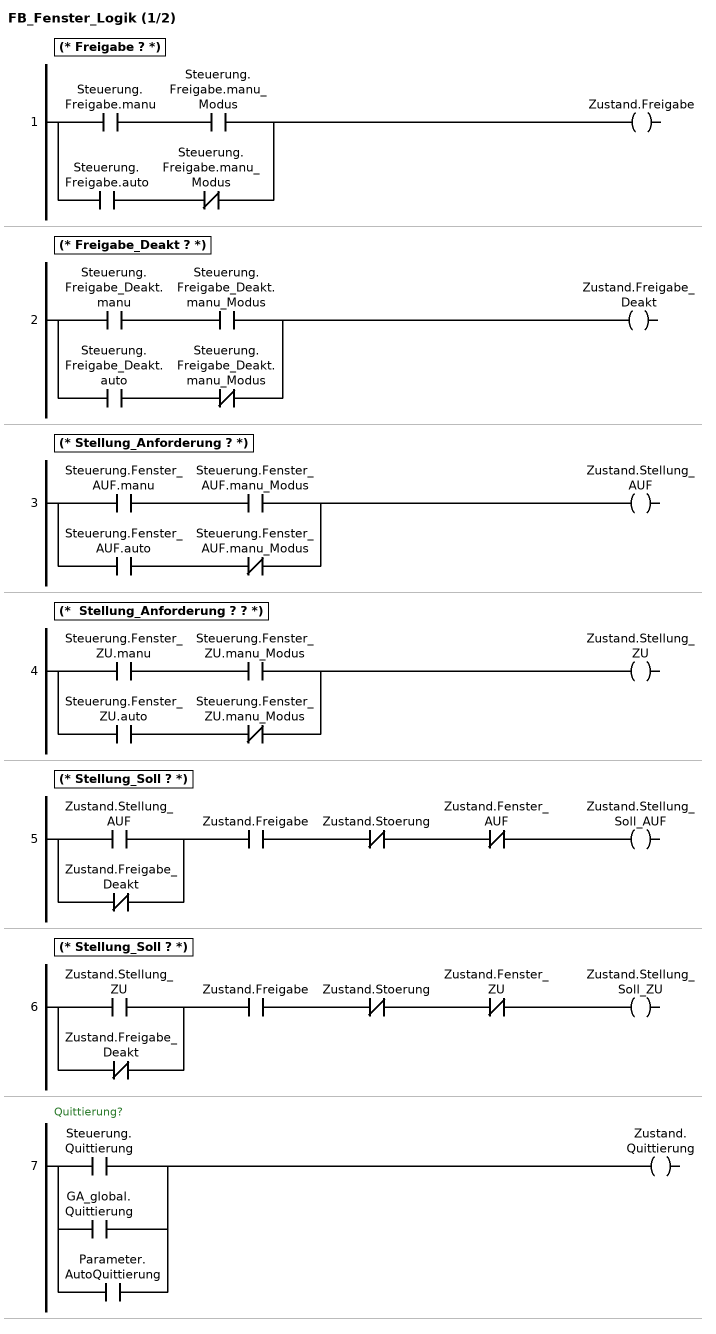
// NETWORK 1
// label: (* Freigabe ? *)
Zustand.Freigabe := Steuerung.Freigabe.manu AND Steuerung.Freigabe.manu_Modus OR Steuerung.Freigabe.auto AND NOT Steuerung.Freigabe.manu_Modus;

// NETWORK 2
// label: (* Freigabe_Deakt ? *)
Zustand.Freigabe_Deakt := Steuerung.Freigabe_Deakt.manu AND Steuerung.Freigabe_Deakt.manu_Modus OR Steuerung.Freigabe_Deakt.auto AND NOT Steuerung.Freigabe_Deakt.manu_Modus;

// NETWORK 3
// label: (* Stellung_Anforderung ? *)
Zustand.Stellung_AUF := Steuerung.Fenster_AUF.manu AND Steuerung.Fenster_AUF.manu_Modus OR Steuerung.Fenster_AUF.auto AND NOT Steuerung.Fenster_AUF.manu_Modus;

// NETWORK 4
// label: (*  Stellung_Anforderung ? ? *)
Zustand.Stellung_ZU := Steuerung.Fenster_ZU.manu AND Steuerung.Fenster_ZU.manu_Modus OR Steuerung.Fenster_ZU.auto AND NOT Steuerung.Fenster_ZU.manu_Modus;

// NETWORK 5
// label: (* Stellung_Soll ? *)
Zustand.Stellung_Soll_AUF := (Zustand.Stellung_AUF OR NOT Zustand.Freigabe_Deakt) AND Zustand.Freigabe AND NOT Zustand.Stoerung AND NOT Zustand.Fenster_AUF;

// NETWORK 6
// label: (* Stellung_Soll ? *)
Zustand.Stellung_Soll_ZU := (Zustand.Stellung_ZU OR NOT Zustand.Freigabe_Deakt) AND Zustand.Freigabe AND NOT Zustand.Stoerung AND NOT Zustand.Fenster_ZU;

// NETWORK 7
// Quittierung?
Zustand.Quittierung := Steuerung.Quittierung OR GA_global.Quittierung OR Parameter.AutoQuittierung;

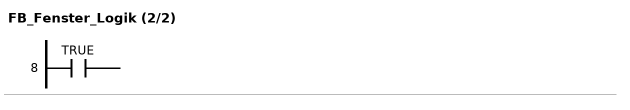
// NETWORK 8

END_FUNCTION_BLOCK

// ---- POUs/Einzelanlagen/RGBW-Kanal/FB_RGBW_Zustandscheck.TcPOU
FUNCTION_BLOCK FB_RGBW_Zustandscheck
VAR_INPUT
	Zustand		: ST_RGBW_Zustand;
	Steuerung	: ST_RGBW_Steuerung;
END_VAR
VAR_OUTPUT
END_VAR
VAR
	RGB_Werte	: ARRAY[0..2] OF BYTE;
	TGB_Werte	: BOOL;
END_VAR

IF Zustand.Betrieb THEN
	HEXSTR_TO_DATA(Steuerung.Farbcode, ADR(RGB_Werte), SIZEOF(RGB_Werte));
	Zustand.R_Wert 	:= RGB_Werte[0];
	Zustand.G_Wert	:= RGB_Werte[1];
	Zustand.B_Wert	:= RGB_Werte[2];
	(*Zustand.W_Wert	:= (0.2126 * ((Zustand.R_Wert / 255) ** 2.2) + 0.7152 * ((Zustand.G_Wert / 255) ** 2.2) + 0.0722 * ((Zustand.B_Wert / 255) ** 2.2));*)
ELSE
	Zustand.R_Wert 	:= 0;
	Zustand.G_Wert	:= 0;
	Zustand.B_Wert	:= 0;
	Zustand.W_Wert	:= 0;
END_IF;

END_FUNCTION_BLOCK

// ---- POUs/Einzelanlagen/Stromzähler/ABB_Stromzaehler/FB_ABB_Lesen.TcPOU
FUNCTION_BLOCK FB_ABB_Lesen
VAR_INPUT
	Reg1Value	: LREAL;
	Reg42Value	: LREAL;
	Reg42Unit 	: STRING;
END_VAR
VAR_OUTPUT
	Arbeit 		: LREAL;
	Leistung 	: LREAL;
	CosPhi		: LREAL;
	(*Scheinleistung: LREAL;
	Blindleistung: LREAL;*)
END_VAR
VAR
	Telegram 	: INT;
END_VAR

(*Der Zähler sendet 5 Versch. Diagramme, es werden jedoch von der Klemme immer nur 2 Diagramme gelesen. Durch prüfen der Einheit des Registers 42 kann bestimmt werden welches Diagramm aktuell gelesen wird.
Reg42.sUnit = 'W' --> Telegram 1+2 werden aktuell ausgelesen
Reg42.sUnit = 'Wh' --> Telegram 3+4 werden aktuell ausgelesen
Reg42.sUnit = '' --> Telegram 5 wird aktuell ausgelesen
*)

IF REG42Unit = 'W' THEN
	Telegram :=1;
ELSIF REG42Unit = 'Wh' THEN
	Telegram :=3;
ELSIF REG42Unit = '' THEN
	Telegram :=5;
END_IF

CASE Telegram OF
	1: 	Arbeit := Reg1Value;
		Leistung := Reg42Value;
	3:	CosPhi := Reg1Value/INT_TO_LREAL(1000);
END_CASE;

(*
(*Scheinleistung berechnen, abfangen von div by 0 error*)
IF  CosPhi<>0  THEN
Scheinleistung := Leistung/CosPhi;
END_IF

(*Blindleistung aus geom Summe berechen, abfangen einer "negativen Wurzel")*)
IF Scheinleistung>Blindleistung THEN
Blindleistung := SQRT(Scheinleistung*Scheinleistung-Leistung*Leistung);
END_IF
*)

END_FUNCTION_BLOCK

// ---- POUs/Einzelanlagen/Stromzähler/ABB_Stromzaehler/FB_Stromzaehler_BHKW.TcPOU
FUNCTION_BLOCK FB_Stromzaehler_BHKW
VAR_INPUT
	Telegramm	: ARRAY[1..cMBUS_MaxTelegrams] OF ST_MBus_Data2;

END_VAR
VAR_IN_OUT
	Zustand		: ST_SZ_Zustand;
END_VAR
VAR
END_VAR
VAR // added by the converter: edge detectors and wires of the graphical bodies
    _w1, _w2 : ANY;
END_VAR

Zustand.Arbeit := _w1;
Zustand.Leistung := _w2;
_w1 := STRING_TO_REAL(Telegramm[1].arrData[1].sValue);
_w2 := STRING_TO_REAL(Telegramm[1].arrData[2].sValue);

END_FUNCTION_BLOCK

// ---- POUs/Einzelanlagen/Stromzähler/ABB_Stromzaehler/FB_Stromzaehler_Gebaeude.TcPOU
FUNCTION_BLOCK FB_Stromzaehler_Gebaeude
VAR_INPUT
	Telegramm	: ARRAY[1..cMBUS_MaxTelegrams] OF ST_MBus_Data2;
END_VAR
VAR_IN_OUT
	Zustand		: ST_SZ_Zustand;
END_VAR
VAR
	Leistungsberechnung			: FB_ABB_Lesen;
END_VAR
VAR // added by the converter: edge detectors and wires of the graphical bodies
    _w1 : ANY;
END_VAR

Zustand.Arbeit := STRING_TO_REAL(Telegramm[1].arrData[1].sValue);
Zustand.Leistung := STRING_TO_REAL(Telegramm[2].arrData[2].sValue);
Zustand.Leistungsfaktor := _w1;
_w1 := STRING_TO_REAL(Telegramm[1].arrData[3].sValue) / 1000;

END_FUNCTION_BLOCK

// ---- POUs/Einzelanlagen/Stromzähler/Netzanschlusspunkt/FB_Stromzaehler_NSHV_Modbus.TcPOU
FUNCTION_BLOCK FB_Stromzaehler_NSHV_Modbus
VAR_IN_OUT
	Stromzaehler_NSHV	: ST_NSHV_Zustand;
END_VAR
VAR_OUTPUT
END_VAR
VAR
	MB_KM				:	ARRAY[1..1] OF ST_NSHV_Modbus;
	ModbusAddress	 	: ARRAY [1..1] OF BYTE := [1]; (*Modbusadressen der beiden Geräte*)
	FtrigBusy			: F_TRIG;
	Timeout 			: TIME := T#300ms;		(* timeout while waiting for an answer of the modbus slave *)
	Unit				: BYTE;
	state				: INT;
	busy				: BOOL;
	LetzterFehlerState	: INT;
	LetzterModbusFehler	: ST_ModbusErrorDiagnostics;
	CounterError		: DINT;
	CounterSuccess		: DINT;
	NSHV_Wert_zuweisen	: FB_NSHV_Wert_zuweisen;
END_VAR

CASE state OF
	0:
		Modbus_NSHV.ReadRegs(Execute:= FALSE); (* Initialisierung*)
		Modbus_NSHV.WriteRegs(Execute:= FALSE);

		(*Auswahl von Modbus-Slaves 1 und 2*)
		Unit := Unit + 1;
		IF Unit  >1 THEN
			Unit := 1;
		END_IF

		state := state + 1;


	1:	(*= NSHV_Spannung_PH1_N lesen =*)
		Modbus_NSHV.ReadRegs(
				UnitID:= ModbusAddress[Unit], (* station address *)
				Quantity:= 2, (*Datenwörter *)
				MBAddr:= 16#1002,
				cbLength:= SIZEOF(MB_KM[Unit].Modbus_Adresse1[16#1002]),
				pMemoryAddr:= ADR(MB_KM[Unit].Modbus_Adresse1[16#1002]),
				Execute:= TRUE,
				Timeout:= Timeout,
				Busy => busy	);
			IF NOT busy THEN
				Modbus_NSHV.ReadRegs(Execute:= FALSE);
				IF Modbus_NSHV.Error THEN
					MB_KM[Unit].Modbus_Unit_Online := FALSE; (*Modbus Gerät ist offline*)
					state := 0;
				ELSE
					MB_KM[Unit].Modbus_Unit_Online := TRUE; (*Modbus Gerät ist online*)
					state := state + 1;
				END_IF
			END_IF


	2:	(*= NSHV_Spannung_PH2_N lesen =*)
		Modbus_NSHV.ReadRegs(
				UnitID:= ModbusAddress[Unit], (* station address *)
				Quantity:= 2, (*Datenwörter *)
				MBAddr:= 16#1004,
				cbLength:= SIZEOF(MB_KM[Unit].Modbus_Adresse1[16#1004]),
				pMemoryAddr:= ADR(MB_KM[Unit].Modbus_Adresse1[16#1004]),
				Execute:= TRUE,
				Timeout:= Timeout,
				Busy => busy	);
			IF NOT busy THEN
				Modbus_NSHV.ReadRegs(Execute:= FALSE);
				IF Modbus_NSHV.Error THEN
					MB_KM[Unit].Modbus_Unit_Online := FALSE; (*Modbus Gerät ist offline*)
					state := 0;
				ELSE
					MB_KM[Unit].Modbus_Unit_Online := TRUE; (*Modbus Gerät ist online*)
					state := state + 1;
				END_IF
			END_IF


	3:	(*= NSHV_Spannung_PH3_N lesen =*)
		Modbus_NSHV.ReadRegs(
				UnitID:= ModbusAddress[Unit], (* station address *)
				Quantity:= 2, (*Datenwörter *)
				MBAddr:= 16#1006,
				cbLength:= SIZEOF(MB_KM[Unit].Modbus_Adresse1[16#1006]),
				pMemoryAddr:= ADR(MB_KM[Unit].Modbus_Adresse1[16#1006]),
				Execute:= TRUE,
				Timeout:= Timeout,
				Busy => busy	);
			IF NOT busy THEN
				Modbus_NSHV.ReadRegs(Execute:= FALSE);
				IF Modbus_NSHV.Error THEN
					MB_KM[Unit].Modbus_Unit_Online := FALSE; (*Modbus Gerät ist offline*)
					state := 0;
				ELSE
					MB_KM[Unit].Modbus_Unit_Online := TRUE; (*Modbus Gerät ist online*)
					state := state + 1;
				END_IF
			END_IF


	4:	(*= NSHV_Strom_PH1 lesen =*)
		Modbus_NSHV.ReadRegs(
				UnitID:= ModbusAddress[Unit], (* station address *)
				Quantity:= 2, (*Datenwörter *)
				MBAddr:= 16#1010,
				cbLength:= SIZEOF(MB_KM[Unit].Modbus_Adresse1[16#1010]),
				pMemoryAddr:= ADR(MB_KM[Unit].Modbus_Adresse1[16#1010]),
				Execute:= TRUE,
				Timeout:= Timeout,
				Busy => busy	);
			IF NOT busy THEN
				Modbus_NSHV.ReadRegs(Execute:= FALSE);
				IF Modbus_NSHV.Error THEN
					MB_KM[Unit].Modbus_Unit_Online := FALSE; (*Modbus Gerät ist offline*)
					state := 0;
				ELSE
					MB_KM[Unit].Modbus_Unit_Online := TRUE; (*Modbus Gerät ist online*)
					state := state + 1;
				END_IF
			END_IF


	5:	(*= NSHV_Strom_PH2 lesen =*)
		Modbus_NSHV.ReadRegs(
				UnitID:= ModbusAddress[Unit], (* station address *)
				Quantity:= 2, (*Datenwörter *)
				MBAddr:= 16#1012,
				cbLength:= SIZEOF(MB_KM[Unit].Modbus_Adresse1[16#1012]),
				pMemoryAddr:= ADR(MB_KM[Unit].Modbus_Adresse1[16#1012]),
				Execute:= TRUE,
				Timeout:= Timeout,
				Busy => busy	);
			IF NOT busy THEN
				Modbus_NSHV.ReadRegs(Execute:= FALSE);
				IF Modbus_NSHV.Error THEN
					MB_KM[Unit].Modbus_Unit_Online := FALSE; (*Modbus Gerät ist offline*)
					state := 0;
				ELSE
					MB_KM[Unit].Modbus_Unit_Online := TRUE; (*Modbus Gerät ist online*)
					state := state + 1;
				END_IF
			END_IF

	6:	(*= NSHV_Strom_PH3 lesen =*)
		Modbus_NSHV.ReadRegs(
				UnitID:= ModbusAddress[Unit], (* station address *)
				Quantity:= 2, (*Datenwörter *)
				MBAddr:= 16#1014,
				cbLength:= SIZEOF(MB_KM[Unit].Modbus_Adresse1[16#1014]),
				pMemoryAddr:= ADR(MB_KM[Unit].Modbus_Adresse1[16#1014]),
				Execute:= TRUE,
				Timeout:= Timeout,
				Busy => busy	);
			IF NOT busy THEN
				Modbus_NSHV.ReadRegs(Execute:= FALSE);
				IF Modbus_NSHV.Error THEN
					MB_KM[Unit].Modbus_Unit_Online := FALSE; (*Modbus Gerät ist offline*)
					state := 0;
				ELSE
					MB_KM[Unit].Modbus_Unit_Online := TRUE; (*Modbus Gerät ist online*)
					state := state + 1;
				END_IF
			END_IF


	7:	(*= NSHV_Wirkleistung lesen =*)
		Modbus_NSHV.ReadRegs(
				UnitID:= ModbusAddress[Unit], (* station address *)
				Quantity:= 2, (*Datenwörter *)
				MBAddr:= 16#102E,
				cbLength:= SIZEOF(MB_KM[Unit].Modbus_Adresse1[16#102E]),
				pMemoryAddr:= ADR(MB_KM[Unit].Modbus_Adresse1[16#102E]),
				Execute:= TRUE,
				Timeout:= Timeout,
				Busy => busy	);
			IF NOT busy THEN
				Modbus_NSHV.ReadRegs(Execute:= FALSE);
				IF Modbus_NSHV.Error THEN
					MB_KM[Unit].Modbus_Unit_Online := FALSE; (*Modbus Gerät ist offline*)
					state := 0;
				ELSE
					MB_KM[Unit].Modbus_Unit_Online := TRUE; (*Modbus Gerät ist online*)
					state := state + 1;
				END_IF
			END_IF

	8:	(*= NSHV_Blindleistung lesen =*)
		Modbus_NSHV.ReadRegs(
				UnitID:= ModbusAddress[Unit], (* station address *)
				Quantity:= 2, (*Datenwörter *)
				MBAddr:= 16#1036,
				cbLength:= SIZEOF(MB_KM[Unit].Modbus_Adresse1[16#1036]),
				pMemoryAddr:= ADR(MB_KM[Unit].Modbus_Adresse1[16#1036]),
				Execute:= TRUE,
				Timeout:= Timeout,
				Busy => busy	);
			IF NOT busy THEN
				Modbus_NSHV.ReadRegs(Execute:= FALSE);
				IF Modbus_NSHV.Error THEN
					MB_KM[Unit].Modbus_Unit_Online := FALSE; (*Modbus Gerät ist offline*)
					state := 0;
				ELSE
					MB_KM[Unit].Modbus_Unit_Online := TRUE; (*Modbus Gerät ist online*)
					state := state + 1;
				END_IF
			END_IF


	9:	(*= NSHV_Scheinleistung lesen =*)
		Modbus_NSHV.ReadRegs(
				UnitID:= ModbusAddress[Unit], (* station address *)
				Quantity:= 2, (*Datenwörter *)
				MBAddr:= 16#1026,
				cbLength:= SIZEOF(MB_KM[Unit].Modbus_Adresse1[16#1026]),
				pMemoryAddr:= ADR(MB_KM[Unit].Modbus_Adresse1[16#1026]),
				Execute:= TRUE,
				Timeout:= Timeout,
				Busy => busy	);
			IF NOT busy THEN
				Modbus_NSHV.ReadRegs(Execute:= FALSE);
				IF Modbus_NSHV.Error THEN
					MB_KM[Unit].Modbus_Unit_Online := FALSE; (*Modbus Gerät ist offline*)
					state := 0;
				ELSE
					MB_KM[Unit].Modbus_Unit_Online := TRUE; (*Modbus Gerät ist online*)
					state := state + 1;
				END_IF
			END_IF

	10:	(*= NSHV_Frequenz lesen =*)
		Modbus_NSHV.ReadRegs(
				UnitID:= ModbusAddress[Unit], (* station address *)
				Quantity:= 2, (*Datenwörter *)
				MBAddr:= 16#1046,
				cbLength:= SIZEOF(MB_KM[Unit].Modbus_Adresse1[16#1046]),
				pMemoryAddr:= ADR(MB_KM[Unit].Modbus_Adresse1[16#1046]),
				Execute:= TRUE,
				Timeout:= Timeout,
				Busy => busy	);
			IF NOT busy THEN
				Modbus_NSHV.ReadRegs(Execute:= FALSE);
				IF Modbus_NSHV.Error THEN
					MB_KM[Unit].Modbus_Unit_Online := FALSE; (*Modbus Gerät ist offline*)
					state := 0;
				ELSE
					MB_KM[Unit].Modbus_Unit_Online := TRUE; (*Modbus Gerät ist online*)
					state := state + 1;
				END_IF
			END_IF

	11:	(*= NSHV_Harmonische_Verzerrung_U_PH1_THD lesen =*)
		Modbus_NSHV.ReadRegs(
				UnitID:= ModbusAddress[Unit], (* station address *)
				Quantity:= 2, (*Datenwörter *)
				MBAddr:= 16#1048,
				cbLength:= SIZEOF(MB_KM[Unit].Modbus_Adresse1[16#1048]),
				pMemoryAddr:= ADR(MB_KM[Unit].Modbus_Adresse1[16#1048]),
				Execute:= TRUE,
				Timeout:= Timeout,
				Busy => busy	);
			IF NOT busy THEN
				Modbus_NSHV.ReadRegs(Execute:= FALSE);
				IF Modbus_NSHV.Error THEN
					MB_KM[Unit].Modbus_Unit_Online := FALSE; (*Modbus Gerät ist offline*)
					state := 0;
				ELSE
					MB_KM[Unit].Modbus_Unit_Online := TRUE; (*Modbus Gerät ist online*)
					state := state + 1;
				END_IF
			END_IF

	12:	(*= NSHV_Harmonische_Verzerrung_U_PH2_THD lesen =*)
		Modbus_NSHV.ReadRegs(
				UnitID:= ModbusAddress[Unit], (* station address *)
				Quantity:= 2, (*Datenwörter *)
				MBAddr:= 16#104A,
				cbLength:= SIZEOF(MB_KM[Unit].Modbus_Adresse1[16#104A]),
				pMemoryAddr:= ADR(MB_KM[Unit].Modbus_Adresse1[16#104A]),
				Execute:= TRUE,
				Timeout:= Timeout,
				Busy => busy	);
			IF NOT busy THEN
				Modbus_NSHV.ReadRegs(Execute:= FALSE);
				IF Modbus_NSHV.Error THEN
					MB_KM[Unit].Modbus_Unit_Online := FALSE; (*Modbus Gerät ist offline*)
					state := 0;
				ELSE
					MB_KM[Unit].Modbus_Unit_Online := TRUE; (*Modbus Gerät ist online*)
					state := state + 1;
				END_IF
			END_IF

	13:	(*= NSHV_Harmonische_Verzerrung_U_PH3_THD lesen =*)
		Modbus_NSHV.ReadRegs(
				UnitID:= ModbusAddress[Unit], (* station address *)
				Quantity:= 2, (*Datenwörter *)
				MBAddr:= 16#104C,
				cbLength:= SIZEOF(MB_KM[Unit].Modbus_Adresse1[16#104C]),
				pMemoryAddr:= ADR(MB_KM[Unit].Modbus_Adresse1[16#104C]),
				Execute:= TRUE,
				Timeout:= Timeout,
				Busy => busy	);
			IF NOT busy THEN
				Modbus_NSHV.ReadRegs(Execute:= FALSE);
				IF Modbus_NSHV.Error THEN
					MB_KM[Unit].Modbus_Unit_Online := FALSE; (*Modbus Gerät ist offline*)
					state := 0;
				ELSE
					MB_KM[Unit].Modbus_Unit_Online := TRUE; (*Modbus Gerät ist online*)
					state := state + 1;
				END_IF
			END_IF

	14:	(*= NSHV_Harmonische_Verzerrung_I_PH1_THD lesen =*)
		Modbus_NSHV.ReadRegs(
				UnitID:= ModbusAddress[Unit], (* station address *)
				Quantity:= 2, (*Datenwörter *)
				MBAddr:= 16#104E,
				cbLength:= SIZEOF(MB_KM[Unit].Modbus_Adresse1[16#104E]),
				pMemoryAddr:= ADR(MB_KM[Unit].Modbus_Adresse1[16#104E]),
				Execute:= TRUE,
				Timeout:= Timeout,
				Busy => busy	);
			IF NOT busy THEN
				Modbus_NSHV.ReadRegs(Execute:= FALSE);
				IF Modbus_NSHV.Error THEN
					MB_KM[Unit].Modbus_Unit_Online := FALSE; (*Modbus Gerät ist offline*)
					state := 0;
				ELSE
					MB_KM[Unit].Modbus_Unit_Online := TRUE; (*Modbus Gerät ist online*)
					state := state + 1;
				END_IF
			END_IF

	15:	(*= NSHV_Harmonische_Verzerrung_I_PH2_THD lesen =*)
		Modbus_NSHV.ReadRegs(
				UnitID:= ModbusAddress[Unit], (* station address *)
				Quantity:= 2, (*Datenwörter *)
				MBAddr:= 16#1050,
				cbLength:= SIZEOF(MB_KM[Unit].Modbus_Adresse1[16#1050]),
				pMemoryAddr:= ADR(MB_KM[Unit].Modbus_Adresse1[16#1050]),
				Execute:= TRUE,
				Timeout:= Timeout,
				Busy => busy	);
			IF NOT busy THEN
				Modbus_NSHV.ReadRegs(Execute:= FALSE);
				IF Modbus_NSHV.Error THEN
					MB_KM[Unit].Modbus_Unit_Online := FALSE; (*Modbus Gerät ist offline*)
					state := 0;
				ELSE
					MB_KM[Unit].Modbus_Unit_Online := TRUE; (*Modbus Gerät ist online*)
					state := state + 1;
				END_IF
			END_IF

	16:	(*= NSHV_Harmonische_Verzerrung_I_PH3_THD lesen =*)
		Modbus_NSHV.ReadRegs(
				UnitID:= ModbusAddress[Unit], (* station address *)
				Quantity:= 2, (*Datenwörter *)
				MBAddr:= 16#1052,
				cbLength:= SIZEOF(MB_KM[Unit].Modbus_Adresse1[16#1052]),
				pMemoryAddr:= ADR(MB_KM[Unit].Modbus_Adresse1[16#1052]),
				Execute:= TRUE,
				Timeout:= Timeout,
				Busy => busy	);
			IF NOT busy THEN
				Modbus_NSHV.ReadRegs(Execute:= FALSE);
				IF Modbus_NSHV.Error THEN
					MB_KM[Unit].Modbus_Unit_Online := FALSE; (*Modbus Gerät ist offline*)
					state := 0;
				ELSE
					MB_KM[Unit].Modbus_Unit_Online := TRUE; (*Modbus Gerät ist online*)
					state := state + 1;
				END_IF
			END_IF

	17:	(*= NSHV_Importierte_Wirkenergie lesen =*)
			Modbus_NSHV.ReadRegs(
					UnitID:= ModbusAddress[Unit], (* station address *)
					Quantity:= 2, (*Datenwörter *)
					MBAddr:= 16#103E,
					cbLength:= SIZEOF(MB_KM[Unit].Modbus_Adresse1[16#103E]),
					pMemoryAddr:= ADR(MB_KM[Unit].Modbus_Adresse1[16#103E]),
					Execute:= TRUE,
					Timeout:= Timeout,
					Busy => busy	);
				IF NOT busy THEN
					Modbus_NSHV.ReadRegs(Execute:= FALSE);
					IF Modbus_NSHV.Error THEN
						MB_KM[Unit].Modbus_Unit_Online := FALSE; (*Modbus Gerät ist offline*)
						state := 0;
					ELSE
						MB_KM[Unit].Modbus_Unit_Online := TRUE; (*Modbus Gerät ist online*)
						state := state + 1;
					END_IF
				END_IF

	18:	(*= NSHV_Exportierte_Wirkenergie lesen =*)
			Modbus_NSHV.ReadRegs(
					UnitID:= ModbusAddress[Unit], (* station address *)
					Quantity:= 2, (*Datenwörter *)
					MBAddr:= 16#1042,
					cbLength:= SIZEOF(MB_KM[Unit].Modbus_Adresse1[16#1042]),
					pMemoryAddr:= ADR(MB_KM[Unit].Modbus_Adresse1[16#1042]),
					Execute:= TRUE,
					Timeout:= Timeout,
					Busy => busy	);
				IF NOT busy THEN
					Modbus_NSHV.ReadRegs(Execute:= FALSE);
					IF Modbus_NSHV.Error THEN
						MB_KM[Unit].Modbus_Unit_Online := FALSE; (*Modbus Gerät ist offline*)
						state := 0;
					ELSE
						MB_KM[Unit].Modbus_Unit_Online := TRUE; (*Modbus Gerät ist online*)
						state := state + 1;
					END_IF
				END_IF

	19:	(*= NSHV_Max_LN_Wirkleistung_Demand lesen =*)
			Modbus_NSHV.ReadRegs(
					UnitID:= ModbusAddress[Unit], (* station address *)
					Quantity:= 2, (*Datenwörter *)
					MBAddr:= 16#1070,
					cbLength:= SIZEOF(MB_KM[Unit].Modbus_Adresse1[16#1070]),
					pMemoryAddr:= ADR(MB_KM[Unit].Modbus_Adresse1[16#1070]),
					Execute:= TRUE,
					Timeout:= Timeout,
					Busy => busy	);
				IF NOT busy THEN
					Modbus_NSHV.ReadRegs(Execute:= FALSE);
					IF Modbus_NSHV.Error THEN
						MB_KM[Unit].Modbus_Unit_Online := FALSE; (*Modbus Gerät ist offline*)
						state := 0;
					ELSE
						MB_KM[Unit].Modbus_Unit_Online := TRUE; (*Modbus Gerät ist online*)
						state := 0;
					END_IF
				END_IF
END_CASE

(*Zählen von erfolgreichen und fehlgeschlagenen Leseversuchen*)
FtrigBusy(CLK:=Modbus_NSHV.BUSY );
IF FtrigBusy.Q THEN
	IF Modbus_NSHV.Error THEN
		LetzterModbusFehler := Modbus_NSHV.ErrorDiagnostics;
		LetzterFehlerState := state;
		CounterError := CounterError + 1;
	ELSE
		CounterSuccess := CounterSuccess + 1;
	END_IF
END_IF

(* Zuweisen der Modbus-Werte zu den Zaehler Variablen *)

NSHV_Wert_zuweisen(Input:= MB_KM[1].Modbus_Adresse1[16#1002], Output => Stromzaehler_NSHV.Spannung_Ph1_N);
NSHV_Wert_zuweisen(Input:= MB_KM[1].Modbus_Adresse1[16#1004], Output => Stromzaehler_NSHV.Spannung_Ph2_N);
NSHV_Wert_zuweisen(Input:= MB_KM[1].Modbus_Adresse1[16#1006], Output => Stromzaehler_NSHV.Spannung_Ph3_N);

NSHV_Wert_zuweisen(Input:= MB_KM[1].Modbus_Adresse1[16#1010], Output => Stromzaehler_NSHV.Strom_Ph1);
NSHV_Wert_zuweisen(Input:= MB_KM[1].Modbus_Adresse1[16#1012], Output => Stromzaehler_NSHV.Strom_Ph2);
NSHV_Wert_zuweisen(Input:= MB_KM[1].Modbus_Adresse1[16#1014], Output => Stromzaehler_NSHV.Strom_Ph3);

NSHV_Wert_zuweisen(Input:= MB_KM[1].Modbus_Adresse1[16#102E], Output => Stromzaehler_NSHV.Wirkleistung);
NSHV_Wert_zuweisen(Input:= MB_KM[1].Modbus_Adresse1[16#1036], Output => Stromzaehler_NSHV.Blindleistung);
NSHV_Wert_zuweisen(Input:= MB_KM[1].Modbus_Adresse1[16#1026], Output => Stromzaehler_NSHV.Scheinleistung);
NSHV_Wert_zuweisen(Input:= MB_KM[1].Modbus_Adresse1[16#1046], Output => Stromzaehler_NSHV.Frequenz);

NSHV_Wert_zuweisen(Input:= MB_KM[1].Modbus_Adresse1[16#1048], Output => Stromzaehler_NSHV.Harmonische_Verzerrung_U_Ph1_THD);
NSHV_Wert_zuweisen(Input:= MB_KM[1].Modbus_Adresse1[16#104A], Output => Stromzaehler_NSHV.Harmonische_Verzerrung_U_Ph2_THD);
NSHV_Wert_zuweisen(Input:= MB_KM[1].Modbus_Adresse1[16#104C], Output => Stromzaehler_NSHV.Harmonische_Verzerrung_U_Ph3_THD );
NSHV_Wert_zuweisen(Input:= MB_KM[1].Modbus_Adresse1[16#104E], Output => Stromzaehler_NSHV.Harmonische_Verzerrung_I_Ph1_THD);
NSHV_Wert_zuweisen(Input:= MB_KM[1].Modbus_Adresse1[16#1050], Output => Stromzaehler_NSHV.Harmonische_Verzerrung_I_Ph2_THD);
NSHV_Wert_zuweisen(Input:= MB_KM[1].Modbus_Adresse1[16#1052], Output => Stromzaehler_NSHV.Harmonische_Verzerrung_I_Ph3_THD);

NSHV_Wert_zuweisen(Input:= MB_KM[1].Modbus_Adresse1[16#103E], Output => Stromzaehler_NSHV.Importierte_Wirkenergie);
NSHV_Wert_zuweisen(Input:= MB_KM[1].Modbus_Adresse1[16#1042], Output => Stromzaehler_NSHV.Exportierte_Wirkenergie);
NSHV_Wert_zuweisen(Input:= MB_KM[1].Modbus_Adresse1[16#1070], Output => Stromzaehler_NSHV.Max_Wirkleistung_Demand_System );



Stromzaehler_NSHV.Stoerung := NOT MB_KM[1].Modbus_Unit_Online;

END_FUNCTION_BLOCK

// ---- POUs/Einzelanlagen/Waermepumpe/FB_WP_Ablaufsteuerung.TcPOU
FUNCTION_BLOCK FB_WP_Ablaufsteuerung
VAR_IN_OUT
	Zustand			: ST_WP_Zustand;
	Stellwert		: ST_WP_Stellwert;
END_VAR
VAR_INPUT
	Steuerung		: ST_WP_Steuerung;
	Parameter		: ST_WP_Parameter;
END_VAR
VAR_OUTPUT
END_VAR
VAR
	Timer			: TON;
END_VAR

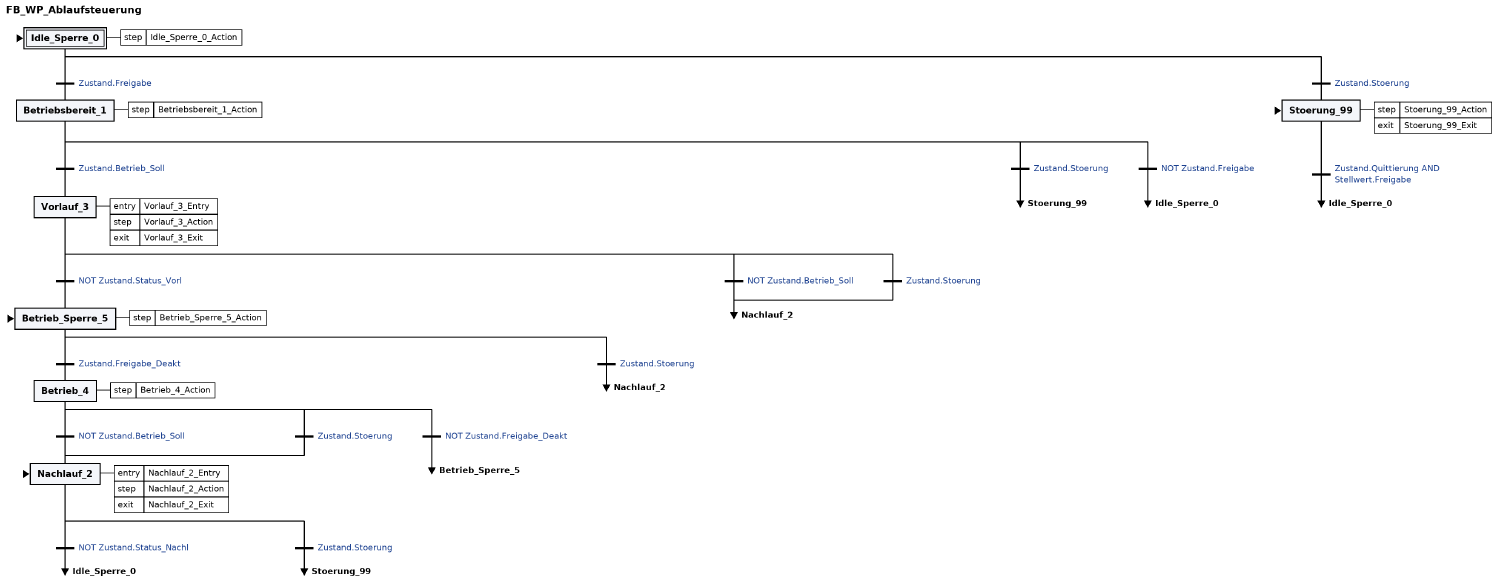
INITIAL_STEP Idle_Sperre_0:
    Idle_Sperre_0_Action(N);  // step action
END_STEP
TRANSITION FROM Idle_Sperre_0 TO Betriebsbereit_1
    := Zustand.Freigabe;
END_TRANSITION
TRANSITION FROM Idle_Sperre_0 TO Stoerung_99
    := Zustand.Stoerung;
END_TRANSITION
STEP Stoerung_99:
    Stoerung_99_Action(N);  // step action
    Stoerung_99_Exit(P0);  // exit action
END_STEP
TRANSITION FROM Stoerung_99 TO Idle_Sperre_0
    := Zustand.Quittierung AND Stellwert.Freigabe;
END_TRANSITION
STEP Betriebsbereit_1:
    Betriebsbereit_1_Action(N);  // step action
END_STEP
TRANSITION FROM Betriebsbereit_1 TO Vorlauf_3
    := Zustand.Betrieb_Soll;
END_TRANSITION
TRANSITION FROM Betriebsbereit_1 TO Stoerung_99
    := Zustand.Stoerung;
END_TRANSITION
TRANSITION FROM Betriebsbereit_1 TO Idle_Sperre_0
    := NOT Zustand.Freigabe;
END_TRANSITION
STEP Vorlauf_3:
    Vorlauf_3_Entry(P1);  // entry action
    Vorlauf_3_Action(N);  // step action
    Vorlauf_3_Exit(P0);  // exit action
END_STEP
TRANSITION FROM Vorlauf_3 TO Betrieb_Sperre_5
    := NOT Zustand.Status_Vorl;
END_TRANSITION
TRANSITION FROM Vorlauf_3 TO Nachlauf_2
    := NOT Zustand.Betrieb_Soll;
END_TRANSITION
TRANSITION FROM Vorlauf_3 TO Nachlauf_2
    := Zustand.Stoerung;
END_TRANSITION
STEP Betrieb_Sperre_5:
    Betrieb_Sperre_5_Action(N);  // step action
END_STEP
TRANSITION FROM Betrieb_Sperre_5 TO Betrieb_4
    := Zustand.Freigabe_Deakt;
END_TRANSITION
TRANSITION FROM Betrieb_Sperre_5 TO Nachlauf_2
    := Zustand.Stoerung;
END_TRANSITION
STEP Betrieb_4:
    Betrieb_4_Action(N);  // step action
END_STEP
TRANSITION FROM Betrieb_4 TO Nachlauf_2
    := NOT Zustand.Betrieb_Soll;
END_TRANSITION
TRANSITION FROM Betrieb_4 TO Nachlauf_2
    := Zustand.Stoerung;
END_TRANSITION
TRANSITION FROM Betrieb_4 TO Betrieb_Sperre_5
    := NOT Zustand.Freigabe_Deakt;
END_TRANSITION
STEP Nachlauf_2:
    Nachlauf_2_Entry(P1);  // entry action
    Nachlauf_2_Action(N);  // step action
    Nachlauf_2_Exit(P0);  // exit action
END_STEP
TRANSITION FROM Nachlauf_2 TO Idle_Sperre_0
    := NOT Zustand.Status_Nachl;
END_TRANSITION
TRANSITION FROM Nachlauf_2 TO Stoerung_99
    := Zustand.Stoerung;
END_TRANSITION

ACTION Betrieb_4_Action:
(* Stellwert setzen *)
Stellwert.Betrieb := TRUE;

(* Zustand setzen *)
Zustand.Status := E_WP_Zustand_Status_Betrieb;
END_ACTION

ACTION Betrieb_Sperre_5_Action:
(* Stellwert setzen *)
Stellwert.Betrieb := TRUE;

(* Zustand setzen *)
Zustand.Status := E_WP_Zustand_Status_Betrieb_Sperre;
END_ACTION

ACTION Betriebsbereit_1_Action:
(* Stellwert setzen *)
Stellwert.Betrieb := FALSE;
Stellwert.Freigabe := TRUE;

(* Zustand setzen *)
Zustand.Status := E_WP_Zustand_Status_Betriebsbereit;
END_ACTION

ACTION Idle_Sperre_0_Action:
(* Stellwert setzen *)
Stellwert.Betrieb := FALSE;

(* Zustand setzen *)
Zustand.Status := E_WP_Zustand_Status_Idle_Sperre;
END_ACTION

ACTION Nachlauf_2_Action:
(* Nachlauf Timer starten *)
Timer( 	IN := Zustand.Status_Nachl,
		PT := DINT_TO_TIME(Parameter.Zeit_Nachl)
);
Zustand.Status_Nachl	:= NOT(Timer.Q AND NOT Zustand.Betrieb);

(* Stellwert setzen *)
Stellwert.Betrieb := FALSE;
Stellwert.Freigabe := FALSE;

(* Zustand setzen *)
Zustand.Status := E_WP_Zustand_Status_Nachl;
END_ACTION

ACTION Nachlauf_2_Entry:
Zustand.Status_Nachl := TRUE;
(* Reset Timer *)
Timer(IN := FALSE);
END_ACTION

ACTION Nachlauf_2_Exit:
Zustand.Status_Nachl := FALSE;
END_ACTION

ACTION Stoerung_99_Action:
(* Stellwert setzen *)
Stellwert.Betrieb := FALSE;

(* Zustand setzen *)
Zustand.Stoerung := TRUE;
Zustand.Status := E_WP_Zustand_Status_Stoerung;
END_ACTION

ACTION Stoerung_99_Exit:
Zustand.Stoerung	:= FALSE;
END_ACTION

ACTION Vorlauf_3_Action:
(* Vorlaufzeit Timer starten *)
Timer( 	IN := Zustand.Status_Vorl,
		PT := DINT_TO_TIME(Parameter.Zeit_Vorl)
);
Zustand.Status_Vorl := NOT (Timer.Q);

(* Stellwert setzen *)
IF Stellwert.Freigabe THEN
	Stellwert.Betrieb := TRUE;
END_IF

(* Zustand setzen *)
Zustand.Status := E_WP_Zustand_Status_Vorl;
END_ACTION

ACTION Vorlauf_3_Entry:
Zustand.Status_Vorl := TRUE;
(* Reset Timer *)
Timer(IN := FALSE);
END_ACTION

ACTION Vorlauf_3_Exit:
Zustand.Status_Vorl := FALSE;
END_ACTION

END_FUNCTION_BLOCK

// ---- POUs/Einzelanlagen/Waermepumpe/FB_WP_Logik.TcPOU
FUNCTION_BLOCK FB_WP_Logik
VAR_IN_OUT
	Steuerung	: ST_WP_Steuerung;
	Zustand		: ST_WP_Zustand;
END_VAR
VAR_INPUT
	Parameter	: ST_WP_Parameter;
END_VAR
VAR_OUTPUT
END_VAR
VAR
END_VAR

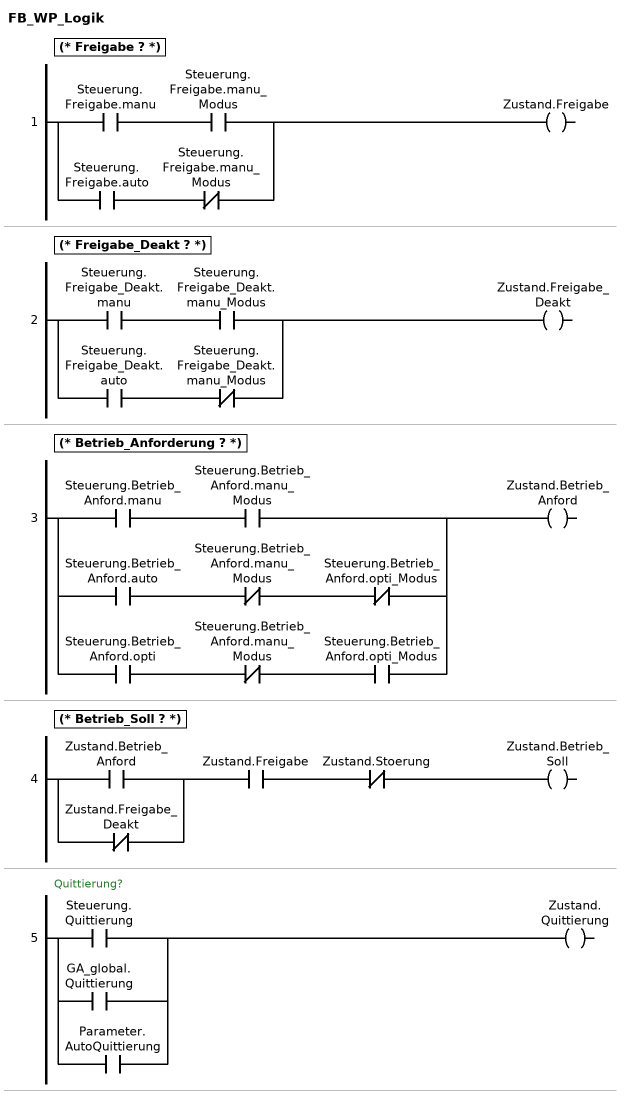
// NETWORK 1
// label: (* Freigabe ? *)
Zustand.Freigabe := Steuerung.Freigabe.manu AND Steuerung.Freigabe.manu_Modus OR Steuerung.Freigabe.auto AND NOT Steuerung.Freigabe.manu_Modus;

// NETWORK 2
// label: (* Freigabe_Deakt ? *)
Zustand.Freigabe_Deakt := Steuerung.Freigabe_Deakt.manu AND Steuerung.Freigabe_Deakt.manu_Modus OR Steuerung.Freigabe_Deakt.auto AND NOT Steuerung.Freigabe_Deakt.manu_Modus;

// NETWORK 3
// label: (* Betrieb_Anforderung ? *)
Zustand.Betrieb_Anford := Steuerung.Betrieb_Anford.manu AND Steuerung.Betrieb_Anford.manu_Modus OR Steuerung.Betrieb_Anford.auto AND NOT Steuerung.Betrieb_Anford.manu_Modus AND NOT Steuerung.Betrieb_Anford.opti_Modus OR Steuerung.Betrieb_Anford.opti AND NOT Steuerung.Betrieb_Anford.manu_Modus AND Steuerung.Betrieb_Anford.opti_Modus;

// NETWORK 4
// label: (* Betrieb_Soll ? *)
Zustand.Betrieb_Soll := (Zustand.Betrieb_Anford OR NOT Zustand.Freigabe_Deakt) AND Zustand.Freigabe AND NOT Zustand.Stoerung;

// NETWORK 5
// Quittierung?
Zustand.Quittierung := Steuerung.Quittierung OR GA_global.Quittierung OR Parameter.AutoQuittierung;

END_FUNCTION_BLOCK

// ---- POUs/Einzelanlagen/Waermepumpe/FB_WP_SchreibeDaten.TcPOU
FUNCTION_BLOCK FB_WP_SchreibeDaten
VAR_INPUT
	WP_Stellung : BOOL;
END_VAR
VAR_OUTPUT
	OUT_WP_Stellung : BOOL;
END_VAR
VAR
END_VAR

OUT_WP_Stellung := WP_Stellung;

END_FUNCTION_BLOCK

// ---- POUs/Einzelanlagen/Waermepumpe/FB_WP_Zustandscheck.TcPOU
FUNCTION_BLOCK FB_WP_Zustandscheck
VAR_IN_OUT
	Zustand		: ST_WP_Zustand;
END_VAR
VAR_INPUT
	Stellwert	 :ST_WP_Stellwert;
	Steuerung	: ST_WP_Steuerung;
	Parameter	: ST_WP_Parameter;
END_VAR
VAR_OUTPUT
END_VAR
VAR
	Timer1			: TON;
	Timer2			: TON;
	Timer3			: TP;
	Timer3verz		: TOF;
	Counter3			: CTU;
	bCounter3Active	: BOOL;
	bTempUeber		: BOOL;
	bWarnung1		: BOOL;
	bWarnung2		: BOOL;
	bWarnung3		: BOOL;
END_VAR

Zustand.Betrieb:= Stellwert.Betrieb;


(*(*
	Stoerung_Code
		0:	Allgemein Störung WP (intern)
		1:	..
		2:	..
		3:
		4:
		5:
		6:
		7:

	Warnung_Code
		0:	Allgemein Warnung WP (intern)
		1:	keine Betriebsrückmeldung
		2:	keine Leistung

	Freigabe_Code
		0:	Freigabe durch Automatik entzogen
		1:	Freigabe durch Manuell entzogen
		2:	Freigabe durch Stoerung entzogen
		3: 	Freigabe durch hohe Einschalthäufigkeiten entzogen
*)
(* Interne Stoerungen / Warnungen *)

(* Warnung - keine Betriebsrückmeldung trotz Betriebsanforderung nach 1 Minute *)
IF (Zustand.Betrieb_Anford <> Zustand.Betrieb) THEN
	bWarnung1	:= TRUE;
ELSE
	bWarnung1	:= FALSE;
END_IF;
Timer1(	IN := bWarnung1,
		PT := T#1M,
		Q => Zustand.Warnung_Code.1
);

(* Warnung - keine Leistung im Betrieb nach 1 Minute *)
IF (Zustand.Leistung <= 0 AND Zustand.Betrieb_Anford = TRUE) THEN
	bWarnung2	:= TRUE;
ELSE
	bWarnung2	:= FALSE;
END_IF;
Timer2(	IN := bWarnung2,
		PT := T#1M,
		Q => Zustand.Warnung_Code.2
);


(* Warnung - Taktbetrieb / hohe Einschaltfrequenzen (3 Anschaltvorgänge pro Stunde) detektiert *)
Timer3(	IN := Zustand.Betrieb,
		PT := T#60M,
		Q => bCounter3Active
);
Counter3(	CU		:= Zustand.Betrieb_Anford,
			RESET	:= NOT bCounter3Active,
			PV		:= 3,
			Q		=> bWarnung3
);
Timer3verz(	IN := bWarnung3,
			PT := T#60M,
			Q => bWarnung3
);


(* ------------------------------------------------------------------- *)
(* Stoermeldung *)
IF Zustand.Stoerung_Code > 0 THEN
	Zustand.Stoerung := TRUE;
(*ELSE - wird nur durch Quittierung gelöscht
	Zustand.Stoerung := FALSE; *)
END_IF;

(* Warnmeldung *)
IF Zustand.Warnung_Code > 0 THEN
	Zustand.Warnung := TRUE;
ELSE
	Zustand.Warnung := FALSE;
END_IF;


(* ----- Freigabe_Code -------- *)
Zustand.Freigabe_Code.0 := NOT(Steuerung.Freigabe.auto);
Zustand.Freigabe_Code.1 := Steuerung.Freigabe.manu_Modus AND NOT Steuerung.Freigabe.manu;
Zustand.Freigabe_Code.2 := Zustand.Stoerung;
Zustand.Freigabe_Code.3 := bWarnung3;

(* Freigabe *)
IF (Zustand.Freigabe_Code > 0 OR NOT Steuerung.Freigabe.auto ) THEN
	Steuerung.Freigabe.auto := FALSE;
ELSE
	Steuerung.Freigabe.auto := TRUE;
END_IF;*)

END_FUNCTION_BLOCK

// ---- POUs/Einzelanlagen/Wetterstation/FB_WS_Konvertierung.TcPOU
FUNCTION_BLOCK FB_WS_Konvertierung
VAR_INPUT
END_VAR
VAR_OUTPUT
	Windgeschwindigkeit_Value	: REAL;
	Aussentemperatur_Value		: REAL;
	Daemmerung_Value			: REAL;
	Regensensor_Value			: BOOL;
END_VAR
VAR
	Group_0_0_1			: EIB_GROUP_ADDR := (MAIN:=0,SUB_MAIN:=0,NUMBER:=1);
	Group_0_0_2			: EIB_GROUP_ADDR := (MAIN:=0,SUB_MAIN:=0,NUMBER:=2);
	Group_0_0_3			: EIB_GROUP_ADDR := (MAIN:=0,SUB_MAIN:=0,NUMBER:=3);
	Group_0_0_4			: EIB_GROUP_ADDR := (MAIN:=0,SUB_MAIN:=0,NUMBER:=4);

	Windgeschwindigkeit	: EIB_2OCTET_FLOAT_REC;
	Temperatur			: EIB_2OCTET_FLOAT_REC;
	Daemmerung			: EIB_2OCTET_FLOAT_REC;
	Regen				: EIB_BIT_REC;
END_VAR

IF(KL_Wetterstation.bReady) THEN
	Windgeschwindigkeit(
		Group_Address := Group_0_0_1,
		strData_Rec := KL_Wetterstation.str_Data_Rec
	);

	Temperatur(
		Group_Address := Group_0_0_2,
		strData_Rec := KL_Wetterstation.str_Data_Rec
	);

	Daemmerung(
		Group_Address := Group_0_0_3,
		strData_Rec := KL_Wetterstation.str_Data_Rec
	);

	Regen(
		Group_Address := Group_0_0_4,
		strData_Rec := KL_Wetterstation.str_Data_Rec
	);

	Windgeschwindigkeit_Value := Windgeschwindigkeit.rData;
	Aussentemperatur_Value := Temperatur.rData;
	Daemmerung_Value := Daemmerung.rData;
	Regensensor_Value := Regen.bData;
END_IF

END_FUNCTION_BLOCK

// ---- POUs/Einzelanlagen/Wetterstation/FB_WS_Mittelung.TcPOU
FUNCTION_BLOCK FB_WS_Mittelung
VAR_INPUT
	Einzelwert				: REAL;
END_VAR
VAR_OUTPUT
	Tagesmittel				: REAL;
END_VAR
VAR
	stParams				: ST_CTRL_MOVING_AVERAGE_PARAMS;
	Moving_Avg 				: FB_CTRL_MOVING_AVERAGE;
	Buffer 					: ARRAY [1..2880] OF REAL;

	fbGetSystemTime			: GETSYSTEMTIME;
	fileTime				: T_FILETIME;


	SystemTimeStruct		: TIMESTRUCT;

	DateTimeNow				: DT;
	initialisiert 			: BOOL := FALSE;
	Initialisierung			: REAL := 12;
	SommerMittel			: REAL := 17;
	WinterMittel			: REAL := 7;

	bSync					: BOOL := FALSE;
END_VAR

(* Finde heraus, ob Winter/Sommer ist und setze entsprechend die Initialisierungstemperatur *)
fbGetSystemTime( timeLoDW=>fileTime.dwLowDateTime, timeHiDW=>fileTime.dwHighDateTime );
DateTimeNow := SYSTEMTIME_TO_DT( TIMESTR:=SystemTimeStruct );
SystemTimeStruct := FILETIME_TO_SYSTEMTIME( fileTime );

IF 5 <= SystemTimeStruct.wMonth AND SystemTimeStruct.wMonth <= 10 THEN
	(* Sommer *)
	Initialisierung := SommerMittel;
ELSE
	(* Winter *)
	Initialisierung := WinterMittel;
END_IF;

(* Parameter definieren - jede Minuten neuen Wert zum Mittel hinzufügen *)
stParams.tCtrlCycleTime := T#1m;
stParams.tTaskCycleTime := T#5ms;
stParams.nSamplesToFilter := 1440; (* 1min*1440=24h *)
stParams.pWorkArray_ADR := ADR(Buffer); (* size 1440*2 *)
stParams.nWorkArray_SIZEOF := SIZEOF(Buffer);

Moving_Avg(
	fIn := Einzelwert,
	fManSyncValue := Initialisierung,
	bSync := bSync,
	eMode := 2,
	bHold := FALSE,
	stParams := stParams,
);

(* initialisieren *)
IF Moving_Avg.bSyncRequest = TRUE THEN
	Tagesmittel := Initialisierung;
ELSE
	Tagesmittel := Moving_Avg.fOut;
END_IF;


IF NOT(initialisiert) THEN
	bSync := TRUE;
	Tagesmittel := Initialisierung;
	initialisiert := TRUE;
END_IF;

END_FUNCTION_BLOCK

// ---- POUs/Einzelanlagen/Wärmezähler/FB_Waermezaehler_MollineC3.TcPOU
FUNCTION_BLOCK FB_Waermezaehler_MollineC3
VAR_INPUT
	Telegramm	: ARRAY[1..cMBUS_MaxTelegrams] OF ST_MBus_Data2;

END_VAR
VAR_IN_OUT
	Zustand		: ST_WZ_Zustand;
END_VAR
VAR
END_VAR
VAR // added by the converter: edge detectors and wires of the graphical bodies
    _w1, _w2 : ANY;
END_VAR

Zustand.Energie := _w1;
//
// arrData[1] = Fabrikationsnummer
// arrData[2] = Gesamt  Wärme Energie  [Wh]
// arrData[3] = Gesamt  Volumen [m3]
// arrData[4] = aktueller Wert Wärme Energie  [kW]
// arrData[5] = maimaler Leistungswert  [kW]
// arrData[6] =  aktueller Wert Volumenstrom  [l/h]
// arrData[7] = maximaler Wert Volumenstrom [l/h]
// arrData[8] = Vorlauftemperatur  [°C]
// arrData[9] = Rücklauftemperatur [°C]
// arrData[10] = Temperaturdifferenz VL - RL[°C]
//
//
//
// Umrechnung von m3 zu Liter
Zustand.Volumen := _w2;
_w1 := STRING_TO_REAL(Telegramm[1].arrData[2].sValue);
Zustand.Temperatur_Vorlauf := STRING_TO_REAL(Telegramm[1].arrData[8].sValue);
Zustand.Temperatur_Ruecklauf := STRING_TO_REAL(Telegramm[1].arrData[9].sValue);
_w2 := STRING_TO_REAL(Telegramm[1].arrData[3].sValue) * 1000;
Zustand.Volumenstrom := STRING_TO_REAL(Telegramm[1].arrData[6].sValue);
Zustand.Leistung := STRING_TO_REAL(Telegramm[1].arrData[4].sValue);
Zustand.Temperatur_Diff := STRING_TO_REAL(Telegramm[1].arrData[10].sValue);

END_FUNCTION_BLOCK

// ---- POUs/Einzelanlagen/Wärmezähler/FB_Waermezaehler_WP.TcPOU
FUNCTION_BLOCK FB_Waermezaehler_WP
VAR_INPUT
	Telegramm	: ARRAY[1..cMBUS_MaxTelegrams] OF ST_MBus_Data2;

END_VAR
VAR_IN_OUT
	Zustand		: ST_WZ_Zustand;
END_VAR
VAR
END_VAR
VAR // added by the converter: edge detectors and wires of the graphical bodies
    _w1, _w2, _w3 : ANY;
END_VAR

Zustand.Energie := _w1;
// 							arrData[1] = Fabrikationsnummer
// arrData[2] = Energie [Wh]
// arrData[6] = Volumen [m3]
// arrData[7] = Laufzeit [Std]
// arrData[9] = Temperatur Vorlauf [°C]
// arrData[10] = Temperatur_Rücklauf [°C]
// arrData[11] = Temperaturdifferenz [°C]
// arrData[12] = Leistung [W]
// arrData[14] = Volumenstrom [m3/h]
//
// Umrechnung von m3 zu Liter
Zustand.Volumen := _w2;
_w1 := STRING_TO_REAL(Telegramm[1].arrData[2].sValue);
Zustand.Temperatur_Vorlauf := STRING_TO_REAL(Telegramm[1].arrData[9].sValue);
Zustand.Temperatur_Ruecklauf := STRING_TO_REAL(Telegramm[1].arrData[10].sValue);
_w2 := STRING_TO_REAL(Telegramm[1].arrData[6].sValue) * 1000;
// Umrechnung von m3/h zu L/h
Zustand.Volumenstrom := _w3;
Zustand.Leistung := STRING_TO_REAL(Telegramm[1].arrData[12].sValue);
Zustand.Temperatur_Diff := STRING_TO_REAL(Telegramm[1].arrData[11].sValue);
_w3 := STRING_TO_REAL(Telegramm[1].arrData[14].sValue) * 1000;

END_FUNCTION_BLOCK

// ---- POUs/Error_Catch.TcPOU
FUNCTION_BLOCK Error_Catch
VAR_INPUT
			Error : BOOL;
			eErrorIN : E_MBus_Error;
END_VAR

VAR
			eError : E_MBus_Error;
END_VAR

IF Error THEN
	eError := eErrorIn;
END_IF

END_FUNCTION_BLOCK

// ---- POUs/Kommunikation/FB_BUFFER_INT_TO_REAL.TcPOU
(* takes an INT and buffers last value if no new value *)

FUNCTION_BLOCK FB_BUFFER_INT_TO_REAL
VAR_INPUT
	raw_input :INT;
END_VAR
VAR_OUTPUT
	real_output :REAL;
END_VAR
VAR
	last_value : REAL;
	temp : DWORD;
END_VAR

temp := INT_TO_DWORD(raw_input);
temp := BE32_TO_HOST(temp);
MEMCPY(ADR(real_output), ADR(temp), SIZEOF(temp));

(* IsFinite prüft auf finitheit und auf NaN *)

IF NOT IsFinite(F_REAL(real_output)) THEN
	real_output := last_value;
ELSE
	last_value := real_output;
END_IF

END_FUNCTION_BLOCK

// ---- POUs/Kommunikation/FB_BUFFER_REAL_TO_REAL.TcPOU
(* takes a REAL and buffers last value if no new value *)

FUNCTION_BLOCK FB_BUFFER_REAL_TO_REAL
VAR_INPUT
	raw_input :REAL;
END_VAR
VAR_OUTPUT
	real_output :REAL;
END_VAR
VAR
	last_value : REAL;
	temp : REAL;
END_VAR

temp := raw_input;
MEMCPY(ADR(real_output), ADR(temp), SIZEOF(temp));

(* IsFinite prüft auf finitheit und auf NaN *)

IF NOT IsFinite(F_REAL(real_output)) THEN
	real_output := last_value;
ELSE
	last_value := real_output;
END_IF

END_FUNCTION_BLOCK

// ---- POUs/Kommunikation/FB_BUFFER_UDINT_TO_REAL.TcPOU
(* converts 4 Bytes into REAL and buffers last value if no new value *)

FUNCTION_BLOCK FB_BUFFER_UDINT_TO_REAL
VAR_INPUT
	raw_input :UDINT;
END_VAR
VAR_OUTPUT
	real_output :REAL;
END_VAR
VAR
	last_value : REAL;
	temp : DWORD;
END_VAR

temp := UDINT_TO_DWORD(raw_input);
temp := BE32_TO_HOST(temp);
MEMCPY(ADR(real_output), ADR(temp), SIZEOF(temp));

(* IsFinite prüft auf finitheit und auf NaN *)

IF NOT IsFinite(F_REAL(real_output)) THEN
	real_output := last_value;
ELSE
	last_value := real_output;
END_IF

END_FUNCTION_BLOCK

// ---- POUs/MBUS_WZaehler.TcPOU
PROGRAM MBUS_WZaehler (* hier wird die Klemme, an welche der M-Bus mit den Zählern angeschlossen ist, alle 10ms aufgerufen *)
VAR
	Komm_Klemme_WZaehler		: FB_MBUSKL6781;
	WMZ331_Brennwerttherme				: FB_MBUS_General_Ext;	(*1*)
	WMZ321_BHKW_1						: FB_MBUS_General_Ext;	(*3*)
	WMZ322_BHKW_2						: FB_MBUS_General_Ext;	(*4*)
	WMZ251_Druckluftkompressor			: FB_MBUS_General_Ext;	(*5*)
	WMZ215_PWT_1						: FB_MBUS_General_Ext;	(*6*)
	WMZ261_Ofenkuehlung_Dichtungen		: FB_MBUS_General_Ext;	(*7*)
	WMZ361_Abwaerme_Ofen_Abgasfackel	: FB_MBUS_General_Ext;	(*8*)
	adrBrennwerttherme				: ST_MBus_SecAdr := (udiIdNumber:=16#00474907);
	adrBHKW_1						: ST_MBus_SecAdr := (udiIdNumber:=16#00470996);
	adrBHKW_2						: ST_MBus_SecAdr := (udiIdNumber:=16#00474904);
	adrDruckluftkompressor			: ST_MBus_SecAdr := (udiIdNumber:=16#00552639);
	adrPWT_1						: ST_MBus_SecAdr := (udiIdNumber:=16#00455395);
	adrOfenkuehlung_Dichtungen		: ST_MBus_SecAdr := (udiIdNumber:=16#00482160);
	adrAbwaerme_Ofen_Abgasfackel	: ST_MBus_SecAdr := (udiIdNumber:=16#00482192);

	fbcatch : 	Error_Catch;
	fbcatch2 : 	Error_Catch;
END_VAR

Komm_Klemme_WZaehler(stComIn := IN_WZaehler, stComOut := OUT_WZaehler, stCom := Komm_MBus_WZaehler); // FB_MBUSKL6781
fbcatch(Error := Komm_Klemme_WZaehler.bError, eErrorIN := Komm_Klemme_WZaehler.eError); // Error_Catch
WMZ331_Brennwerttherme(usiAddress := 253, stSecAdr := adrBrennwerttherme, stCom := Komm_MBus_WZaehler); // FB_MBUS_General_Ext
Telegramm_WZ_Brennwerttherme := WMZ331_Brennwerttherme.arrTelegram;
WMZ321_BHKW_1(usiAddress := 253, stSecAdr := adrBHKW_1, stCom := Komm_MBus_WZaehler); // FB_MBUS_General_Ext
Telegramm_WZ_BHKW_1 := WMZ321_BHKW_1.arrTelegram;
WMZ322_BHKW_2(usiAddress := 253, stSecAdr := adrBHKW_2, stCom := Komm_MBus_WZaehler); // FB_MBUS_General_Ext
WMZ251_Druckluftkompressor(
    usiAddress := 253,
    stSecAdr := adrDruckluftkompressor,
    stCom := Komm_MBus_WZaehler); // FB_MBUS_General_Ext
WMZ215_PWT_1(usiAddress := 253, stSecAdr := adrPWT_1, stCom := Komm_MBus_WZaehler); // FB_MBUS_General_Ext
WMZ261_Ofenkuehlung_Dichtungen(
    usiAddress := 253,
    stSecAdr := adrOfenkuehlung_Dichtungen,
    stCom := Komm_MBus_WZaehler); // FB_MBUS_General_Ext
Telegramm_WZ_Ofenkuehlung := WMZ261_Ofenkuehlung_Dichtungen.arrTelegram;
WMZ361_Abwaerme_Ofen_Abgasfackel(
    usiAddress := 253,
    stSecAdr := adrAbwaerme_Ofen_Abgasfackel,
    stCom := Komm_MBus_WZaehler); // FB_MBUS_General_Ext
Telegramm_WZ_Abwaerme_Ofen_Abgasfackel := WMZ361_Abwaerme_Ofen_Abgasfackel.arrTelegram;
Telegramm_WZ_BHKW_2 := WMZ322_BHKW_2.arrTelegram;
Telegramm_WZ_Druckluftkompressor := WMZ251_Druckluftkompressor.arrTelegram;
Telegramm_WZ_PWT_1 := WMZ215_PWT_1.arrTelegram;
fbcatch(Error := WMZ331_Brennwerttherme.bError, eErrorIN := WMZ331_Brennwerttherme.eError); // Error_Catch

END_PROGRAM

// ---- POUs/P_EIB.TcPOU
PROGRAM P_EIB
VAR
	fbKL6301				: KL6301;
	grpAdr					: EIB_GROUP_ADDR := (MAIN:=0, SUB_MAIN:=0, NUMBER:=1);
	KL_Wetterstation_IN_1		AT%I*	: ARRAY[1..24]OF BYTE;
	KL_Wetterstation_OUT_1		AT%Q*		: ARRAY[1..24]OF BYTE;
	stDataRec              : EIB_REC;
END_VAR



fbKL6301(
	bActivate:= TRUE,
	idx:= 1,
	EIB_PHYS_ADDR:= grpAdr,
	EIB_GROUP_FILTER:= ,
	iMode:= ,
	KL6301_IN:= KL_Wetterstation_IN_1,
	KL6301_OUT:= KL_Wetterstation_OUT_1,
	bActive=> ,
	bReady=> , 
	bError=> , 
	iErrorId=> , 
	str_Data_Rec=> stDataRec);




EIB_2OCTET_FLOAT_REC(
	Group_Address:= ,
	strData_Rec:= stDataRec,
	bDataReceive=> ,
	rData=> );

END_PROGRAM

// ---- POUs/Systeme/Sonstiges/Beleuchtung/Beleuchtung Außen/FB_System_BelAu.TcPOU
FUNCTION_BLOCK FB_System_BelAu
VAR_INPUT
	Freigabe_auto			: BOOL;
	Betrieb_Anford_auto		: BOOL:= TRUE;
	Regelung_Sollw_auto		: REAL;
	AdressType				: E_DALIV2AddrType;
END_VAR
VAR_OUTPUT
	{attribute 'OPC.UA.DA' := '1'}Steuerung				: ST_System_Bel_Steuerung;		
	{attribute 'OPC.UA.DA' := '1'}Stellwert				: ST_System_Bel_Stellwert;		
	{attribute 'OPC.UA.DA' := '1'}Zustand					: ST_System_Bel_Zustand;	
	{attribute 'OPC.UA.DA' := '1'}Parameter				: ST_System_Bel_Parameter;		
END_VAR
VAR
	Ablaufsteuerung			: FB_System_BelAu_Ablaufsteuerung;
	Regelung				: FB_System_BelAu_Regelung;
	Zustandscheck			: FB_System_BelAu_Zustandscheck;
	SensorikHelligkeit		: FB_System_BelAu_Sensorik;
	Logik 					: FB_System_BelAu_Logik;
	Sollwertscheck			: FB_System_BelAu_Sollwertscheck;
	Stellwertscheck			: FB_System_BelAu_Stellwertscheck;
	Regelung_Modus_auto		: SINT;


	Beleuchtung_NO: FB_Bel_RGBW;
	Beleuchtung_NW: FB_Bel_RGBW;
	Beleuchtung_SO: FB_Bel_RGBW;
	Beleuchtung_SW: FB_Bel_RGBW;
	Beleuchtung_SD: FB_Bel_RGBW;
	Beleuchtung_ND: FB_Bel_RGBW;
	Hex_Farbe	: STRING;
	Farbwert_NO: STRING;
	Farbwert_NW: STRING;
	Farbwert_ND: STRING;
	Farbwert_SO: STRING;
	Farbwert_SW: STRING;
	Farbwert_SD: STRING;


	Reset_NO: TON;
	Reset_NW: TON;
	Reset_ND: TON;
	Reset_SO: TON;
	Reset_SW: TON;
	Reset_SD: TON;
	reset: BOOL;
END_VAR

Farbwert_SW := Regelung.Steuerung_Farbcode_SW;
Farbwert_SD := Regelung.Steuerung_Farbcode_SD;
Beleuchtung_NO(
    Freigabe_auto := Zustand.Freigabe,
    Freigabe_Deakt_auto := Zustand.Freigabe_Deakt,
    Betrieb_Anford_auto := zustand.Betrieb_Anford,
    Farbcode := Farbwert_NO,
    Adresse_R := 40,
    Adresse_G := 41,
    Adresse_B := 42,
    Adresse_W := 43,
    Quittierung := zustand.Quittierung,
    AdressType := eDALIV2AddrTypeGroup,
    Reset := Reset_NO.Q); // FB_Bel_RGBW
Beleuchtung_NW(
    Freigabe_auto := Zustand.Freigabe,
    Freigabe_Deakt_auto := Zustand.Freigabe_Deakt,
    Betrieb_Anford_auto := zustand.Betrieb_Anford,
    Farbcode := Farbwert_NW,
    Adresse_R := 48,
    Adresse_G := 49,
    Adresse_B := 50,
    Adresse_W := 51,
    Quittierung := zustand.Quittierung,
    AdressType := eDALIV2AddrTypeGroup,
    Reset := Reset_NW.Q); // FB_Bel_RGBW
Beleuchtung_SO(
    Freigabe_auto := Zustand.Freigabe,
    Freigabe_Deakt_auto := Zustand.Freigabe_Deakt,
    Betrieb_Anford_auto := zustand.Betrieb_Anford,
    Farbcode := Farbwert_SO,
    Adresse_R := 60,
    Adresse_G := 61,
    Adresse_B := 62,
    Adresse_W := 63,
    Quittierung := zustand.Quittierung,
    AdressType := eDALIV2AddrTypeGroup,
    Reset := Reset_SO.Q); // FB_Bel_RGBW
Beleuchtung_SW(
    Freigabe_auto := Zustand.Freigabe,
    Freigabe_Deakt_auto := Zustand.Freigabe_Deakt,
    Betrieb_Anford_auto := zustand.Betrieb_Anford,
    Farbcode := Farbwert_SW,
    Adresse_R := 52,
    Adresse_G := 53,
    Adresse_B := 54,
    Adresse_W := 55,
    Quittierung := zustand.Quittierung,
    AdressType := eDALIV2AddrTypeGroup,
    Reset := Reset_SW.Q); // FB_Bel_RGBW
Steuerung.Freigabe.auto := Freigabe_auto;
Parameter := Initialisierung.System_Bel_Parameter;
Steuerung.Freigabe_Deakt.auto := TRUE;
Steuerung.Betrieb_Anford.auto := Betrieb_Anford_auto;
Steuerung.Regelung_Sollw.auto := Regelung_Sollw_auto;
Zustandscheck(Steuerung := Steuerung, Parameter := Parameter, Zustand := Zustand); // FB_System_BelAu_Zustandscheck
Logik(Parameter := Parameter, Steuerung := Steuerung, Zustand := Zustand); // FB_System_BelAu_Logik
Ablaufsteuerung(Steuerung := Steuerung, Parameter := Parameter, Zustand := Zustand, Stellwert := Stellwert); // FB_System_BelAu_Ablaufsteuerung
Farbwert_NO := Regelung.Steuerung_Farbcode_NO;
SensorikHelligkeit(); // FB_System_BelAu_Sensorik
Regelung(
    Dunkelheits_Sensor_1 := SensorikHelligkeit.Dunkelheit_OUT,
    Stellwert := Stellwert,
    Steuerung := Steuerung,
    Zustand := Zustand); // FB_System_BelAu_Regelung
Farbwert_NW := Regelung.Steuerung_Farbcode_NW;
Farbwert_ND := Regelung.Steuerung_Farbcode_ND;
Farbwert_SO := Regelung.Steuerung_Farbcode_SO;
Steuerung.Regelung_Modus.auto := Regelung_Modus_auto;
Beleuchtung_SD(
    Freigabe_auto := Zustand.Freigabe,
    Freigabe_Deakt_auto := Zustand.Freigabe_Deakt,
    Betrieb_Anford_auto := zustand.Betrieb_Anford,
    Farbcode := Farbwert_SD,
    Adresse_R := 56,
    Adresse_G := 57,
    Adresse_B := 58,
    Adresse_W := 59,
    Quittierung := zustand.Quittierung,
    AdressType := eDALIV2AddrTypeGroup,
    Reset := Reset_SD.Q); // FB_Bel_RGBW
Beleuchtung_ND(
    Freigabe_auto := Zustand.Freigabe,
    Freigabe_Deakt_auto := Zustand.Freigabe_Deakt,
    Betrieb_Anford_auto := zustand.Betrieb_Anford,
    Farbcode := Farbwert_ND,
    Adresse_R := 44,
    Adresse_G := 45,
    Adresse_B := 46,
    Adresse_W := 47,
    Quittierung := zustand.Quittierung,
    AdressType := eDALIV2AddrTypeGroup,
    Reset := Reset_ND.Q); // FB_Bel_RGBW
Reset_NO(IN := Steuerung.Reset, PT := t#3s); // TON
Reset_NW(IN := Steuerung.Reset, PT := t#4s); // TON
Reset_ND(IN := Steuerung.Reset, PT := t#5s); // TON
Reset_SO(IN := Steuerung.Reset, PT := t#6s); // TON
Reset_SW(IN := Steuerung.Reset, PT := t#7s); // TON
Reset_SD(IN := Steuerung.Reset, PT := t#8s); // TON

END_FUNCTION_BLOCK

// ---- POUs/Systeme/Sonstiges/Beleuchtung/Beleuchtung Außen/FB_System_BelAu_Ablaufsteuerung.TcPOU
FUNCTION_BLOCK FB_System_BelAu_Ablaufsteuerung
VAR_IN_OUT
	Zustand			: ST_System_Bel_Zustand;
	Stellwert		: ST_System_Bel_Stellwert;
END_VAR
VAR_INPUT
	Steuerung		: ST_System_Bel_Steuerung;
	Parameter		: ST_System_Bel_Parameter;
END_VAR
VAR_OUTPUT
END_VAR
VAR
	Timer: TON;
END_VAR

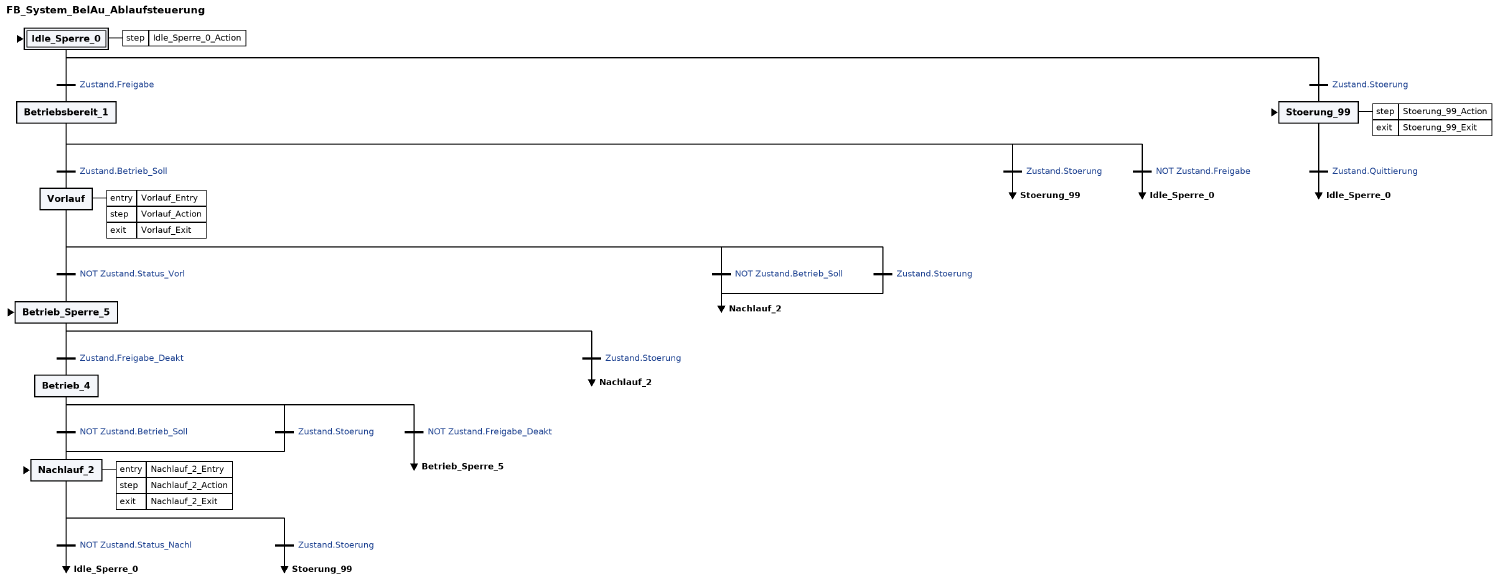
INITIAL_STEP Idle_Sperre_0:
    Idle_Sperre_0_Action(N);  // step action
END_STEP
TRANSITION FROM Idle_Sperre_0 TO Betriebsbereit_1
    := Zustand.Freigabe;
END_TRANSITION
TRANSITION FROM Idle_Sperre_0 TO Stoerung_99
    := Zustand.Stoerung;
END_TRANSITION
STEP Stoerung_99:
    Stoerung_99_Action(N);  // step action
    Stoerung_99_Exit(P0);  // exit action
END_STEP
TRANSITION FROM Stoerung_99 TO Idle_Sperre_0
    := Zustand.Quittierung;
END_TRANSITION
STEP Betriebsbereit_1:
END_STEP
TRANSITION FROM Betriebsbereit_1 TO Vorlauf
    := Zustand.Betrieb_Soll;
END_TRANSITION
TRANSITION FROM Betriebsbereit_1 TO Stoerung_99
    := Zustand.Stoerung;
END_TRANSITION
TRANSITION FROM Betriebsbereit_1 TO Idle_Sperre_0
    := NOT Zustand.Freigabe;
END_TRANSITION
STEP Vorlauf:
    Vorlauf_Entry(P1);  // entry action
    Vorlauf_Action(N);  // step action
    Vorlauf_Exit(P0);  // exit action
END_STEP
TRANSITION FROM Vorlauf TO Betrieb_Sperre_5
    := NOT Zustand.Status_Vorl;
END_TRANSITION
TRANSITION FROM Vorlauf TO Nachlauf_2
    := NOT Zustand.Betrieb_Soll;
END_TRANSITION
TRANSITION FROM Vorlauf TO Nachlauf_2
    := Zustand.Stoerung;
END_TRANSITION
STEP Betrieb_Sperre_5:
END_STEP
TRANSITION FROM Betrieb_Sperre_5 TO Betrieb_4
    := Zustand.Freigabe_Deakt;
END_TRANSITION
TRANSITION FROM Betrieb_Sperre_5 TO Nachlauf_2
    := Zustand.Stoerung;
END_TRANSITION
STEP Betrieb_4:
END_STEP
TRANSITION FROM Betrieb_4 TO Nachlauf_2
    := NOT Zustand.Betrieb_Soll;
END_TRANSITION
TRANSITION FROM Betrieb_4 TO Nachlauf_2
    := Zustand.Stoerung;
END_TRANSITION
TRANSITION FROM Betrieb_4 TO Betrieb_Sperre_5
    := NOT Zustand.Freigabe_Deakt;
END_TRANSITION
STEP Nachlauf_2:
    Nachlauf_2_Entry(P1);  // entry action
    Nachlauf_2_Action(N);  // step action
    Nachlauf_2_Exit(P0);  // exit action
END_STEP
TRANSITION FROM Nachlauf_2 TO Idle_Sperre_0
    := NOT Zustand.Status_Nachl;
END_TRANSITION
TRANSITION FROM Nachlauf_2 TO Stoerung_99
    := Zustand.Stoerung;
END_TRANSITION

ACTION Idle_Sperre_0_Action:
(* Quittierungszustand auf False setzen, damit das System bei einer erneuten Störung nicht direkt wieder angeschaltet wird *)
Steuerung.Quittierung	:= FALSE;
END_ACTION

ACTION Nachlauf_2_Action:
(* Nachlauf Timer starten *)
Timer( 	IN := Zustand.Status_Nachl,
		PT := DINT_TO_TIME(Parameter.Zeit_Nachl)
);
Zustand.Status_Nachl	:= NOT(Timer.Q AND NOT Zustand.Betrieb);

(* Stellwert setzen *)
Stellwert.Betrieb := FALSE;

(* Zustand setzen *)
Zustand.Status := E_Bel_Zustand_Status_Nachl;
END_ACTION

ACTION Nachlauf_2_Entry:
Zustand.Status_Nachl := TRUE;
(* Reset Timer *)
Timer(IN := FALSE);
END_ACTION

ACTION Nachlauf_2_Exit:
Zustand.Status_Nachl := FALSE;
END_ACTION

ACTION Stoerung_99_Action:
(* Stellwert setzen *)
Stellwert.Betrieb := FALSE;

(* Zustand setzen *)
Zustand.Stoerung := TRUE;
Zustand.Status := E_Bel_Zustand_Status_Stoerung;
END_ACTION

ACTION Stoerung_99_Exit:
Zustand.Stoerung	:= FALSE;
END_ACTION

ACTION Vorlauf_Action:
(* Vorlaufzeit Timer starten *)
Timer( 	IN := Zustand.Status_Vorl,
		PT := DINT_TO_TIME(Parameter.Zeit_Vorl)
);
Zustand.Status_Vorl := NOT (Timer.Q AND Zustand.Betrieb);

(* Stellwert setzen *)
Stellwert.Betrieb := TRUE;

(* Zustand setzen *)
Zustand.Status := E_Bel_Zustand_Status_Vorl;
END_ACTION

ACTION Vorlauf_Entry:
Zustand.Status_Vorl := TRUE;
(* Reset Timer *)
Timer(IN := FALSE);
END_ACTION

ACTION Vorlauf_Exit:
Zustand.Status_Vorl := FALSE;
END_ACTION

END_FUNCTION_BLOCK

// ---- POUs/Systeme/Sonstiges/Beleuchtung/Beleuchtung Außen/FB_System_BelAu_Logik.TcPOU
FUNCTION_BLOCK FB_System_BelAu_Logik
VAR_IN_OUT
	Steuerung	: ST_System_Bel_Steuerung;
	Zustand		: ST_System_Bel_Zustand;
END_VAR
VAR_INPUT
	Parameter	: ST_System_Bel_Parameter;
END_VAR
VAR_OUTPUT
END_VAR
VAR
END_VAR

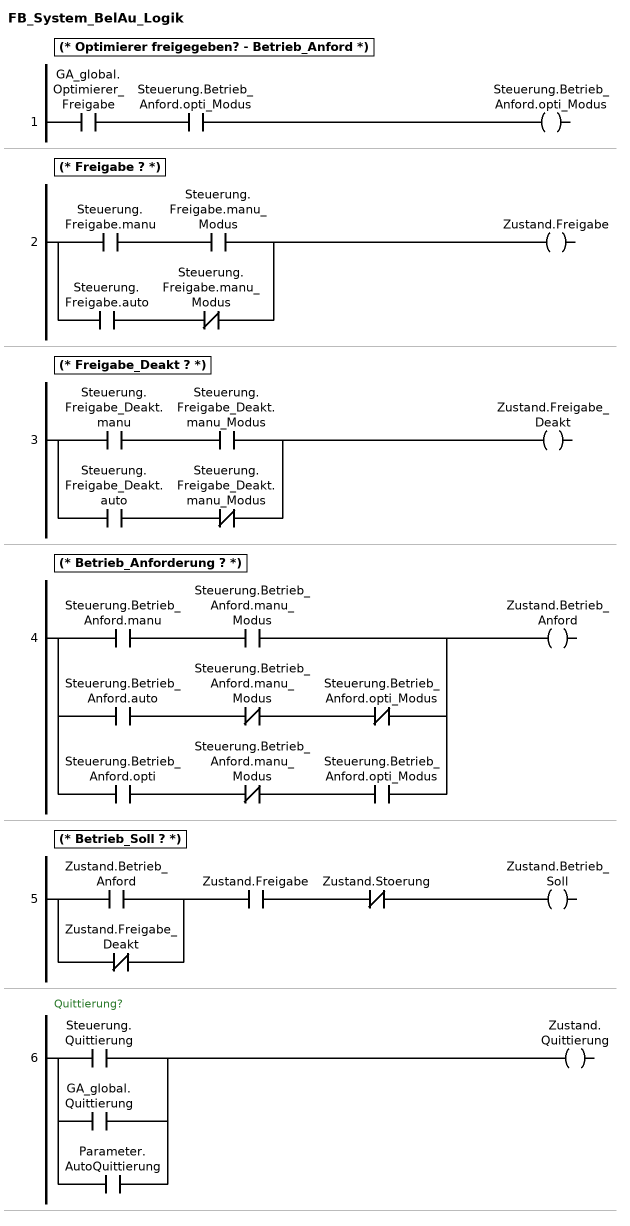
// NETWORK 1
// label: (* Optimierer freigegeben? - Betrieb_Anford *)
Steuerung.Betrieb_Anford.opti_Modus := GA_global.Optimierer_Freigabe AND Steuerung.Betrieb_Anford.opti_Modus;

// NETWORK 2
// label: (* Freigabe ? *)
Zustand.Freigabe := Steuerung.Freigabe.manu AND Steuerung.Freigabe.manu_Modus OR Steuerung.Freigabe.auto AND NOT Steuerung.Freigabe.manu_Modus;

// NETWORK 3
// label: (* Freigabe_Deakt ? *)
Zustand.Freigabe_Deakt := Steuerung.Freigabe_Deakt.manu AND Steuerung.Freigabe_Deakt.manu_Modus OR Steuerung.Freigabe_Deakt.auto AND NOT Steuerung.Freigabe_Deakt.manu_Modus;

// NETWORK 4
// label: (* Betrieb_Anforderung ? *)
Zustand.Betrieb_Anford := Steuerung.Betrieb_Anford.manu AND Steuerung.Betrieb_Anford.manu_Modus OR Steuerung.Betrieb_Anford.auto AND NOT Steuerung.Betrieb_Anford.manu_Modus AND NOT Steuerung.Betrieb_Anford.opti_Modus OR Steuerung.Betrieb_Anford.opti AND NOT Steuerung.Betrieb_Anford.manu_Modus AND Steuerung.Betrieb_Anford.opti_Modus;

// NETWORK 5
// label: (* Betrieb_Soll ? *)
Zustand.Betrieb_Soll := (Zustand.Betrieb_Anford OR NOT Zustand.Freigabe_Deakt) AND Zustand.Freigabe AND NOT Zustand.Stoerung;

// NETWORK 6
// Quittierung?
Zustand.Quittierung := Steuerung.Quittierung OR GA_global.Quittierung OR Parameter.AutoQuittierung;

END_FUNCTION_BLOCK

// ---- POUs/Systeme/Sonstiges/Beleuchtung/Beleuchtung Außen/FB_System_BelAu_Sollwertscheck.TcPOU
FUNCTION_BLOCK FB_System_BelAu_Sollwertscheck
VAR_IN_OUT
	Zustand		: ST_System_Bel_Zustand;
END_VAR
VAR_INPUT
	Steuerung	: ST_System_Bel_Steuerung;
END_VAR
VAR
END_VAR

(* Priorisierung Regelung_Modus *)
IF(Steuerung.Regelung_Modus.manu_Modus) THEN
	Zustand.Regelung_Modus := Steuerung.Regelung_Modus.manu;
ELSIF(Steuerung.Regelung_Modus.opti_Modus) THEN
	Zustand.Regelung_Modus := Steuerung.Regelung_Modus.opti;
ELSE
	Zustand.Regelung_Modus := Steuerung.Regelung_Modus.auto;
END_IF;
(* Priorisierung Regelung_Sollwert *)
IF(Steuerung.Regelung_Sollw.manu_Modus) THEN
	Zustand.Regelung_Sollw := Steuerung.Regelung_Sollw.manu;
ELSIF(Steuerung.Regelung_Sollw.opti_Modus) THEN
	Zustand.Regelung_Sollw := Steuerung.Regelung_Sollw.opti;
ELSE
	Zustand.Regelung_Sollw := Steuerung.Regelung_Sollw.auto;
END_IF;
(*IF (Zustand.Regelung_Modus_Anford )THEN
	Zustand.Regelung_Modus  :=E_Bel_Regelung_Modus_Lichtsensor ;
ELSE
	Zustand.Regelung_Modus := E_Bel_Regelung_Modus_P ;
END_IF*)

END_FUNCTION_BLOCK

// ---- POUs/Systeme/Sonstiges/Beleuchtung/Beleuchtung Halle/FB_System_BelHa_Logik.TcPOU
FUNCTION_BLOCK FB_System_BelHa_Logik
VAR_IN_OUT
	Steuerung	: ST_System_Bel_Steuerung;
	Zustand		: ST_System_Bel_Zustand;
END_VAR
VAR_INPUT
	Parameter	: ST_System_Bel_Parameter;
END_VAR
VAR_OUTPUT
END_VAR
VAR
END_VAR

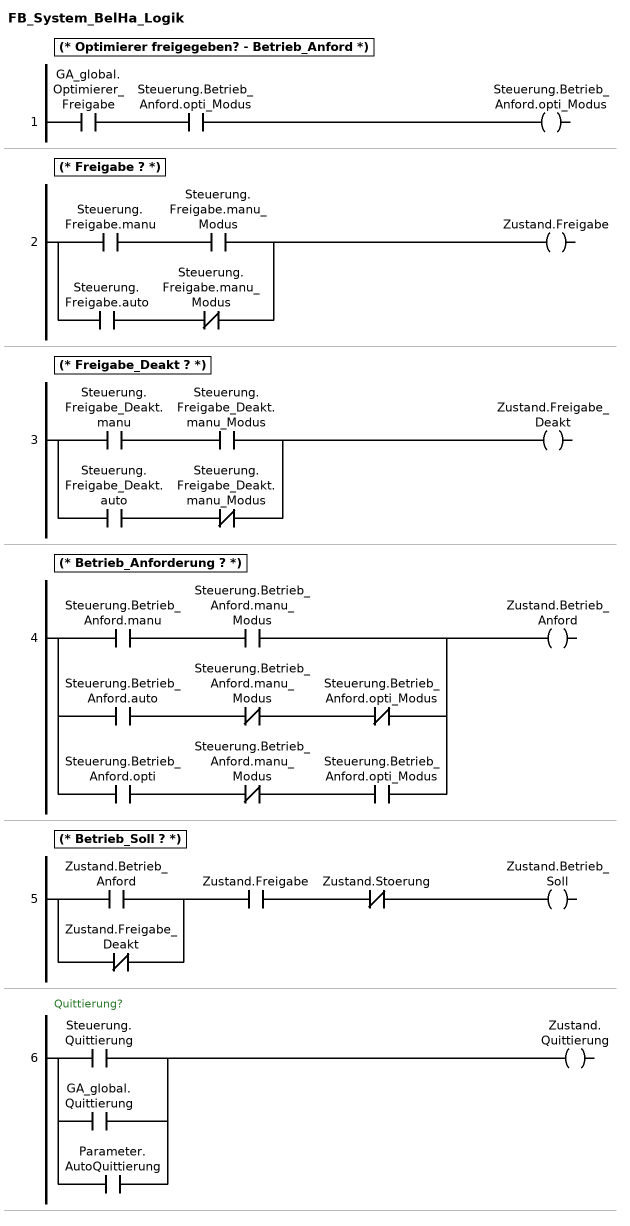
// NETWORK 1
// label: (* Optimierer freigegeben? - Betrieb_Anford *)
Steuerung.Betrieb_Anford.opti_Modus := GA_global.Optimierer_Freigabe AND Steuerung.Betrieb_Anford.opti_Modus;

// NETWORK 2
// label: (* Freigabe ? *)
Zustand.Freigabe := Steuerung.Freigabe.manu AND Steuerung.Freigabe.manu_Modus OR Steuerung.Freigabe.auto AND NOT Steuerung.Freigabe.manu_Modus;

// NETWORK 3
// label: (* Freigabe_Deakt ? *)
Zustand.Freigabe_Deakt := Steuerung.Freigabe_Deakt.manu AND Steuerung.Freigabe_Deakt.manu_Modus OR Steuerung.Freigabe_Deakt.auto AND NOT Steuerung.Freigabe_Deakt.manu_Modus;

// NETWORK 4
// label: (* Betrieb_Anforderung ? *)
Zustand.Betrieb_Anford := Steuerung.Betrieb_Anford.manu AND Steuerung.Betrieb_Anford.manu_Modus OR Steuerung.Betrieb_Anford.auto AND NOT Steuerung.Betrieb_Anford.manu_Modus AND NOT Steuerung.Betrieb_Anford.opti_Modus OR Steuerung.Betrieb_Anford.opti AND NOT Steuerung.Betrieb_Anford.manu_Modus AND Steuerung.Betrieb_Anford.opti_Modus;

// NETWORK 5
// label: (* Betrieb_Soll ? *)
Zustand.Betrieb_Soll := (Zustand.Betrieb_Anford OR NOT Zustand.Freigabe_Deakt) AND Zustand.Freigabe AND NOT Zustand.Stoerung;

// NETWORK 6
// Quittierung?
Zustand.Quittierung := Steuerung.Quittierung OR GA_global.Quittierung OR Parameter.AutoQuittierung;

END_FUNCTION_BLOCK

// ---- POUs/Systeme/Sonstiges/Beleuchtung/Beleuchtung Halle/FB_System_BelHa_Sollwertscheck.TcPOU
FUNCTION_BLOCK FB_System_BelHa_Sollwertscheck
VAR_IN_OUT
	Zustand		: ST_System_Bel_Zustand;
END_VAR
VAR_INPUT
	Steuerung	: ST_System_Bel_Steuerung;
END_VAR
VAR
END_VAR

(* Priorisierung Regelung_Modus *)
IF(Steuerung.Regelung_Modus.manu_Modus) THEN
	Zustand.Regelung_Modus := Steuerung.Regelung_Modus.manu;
ELSIF(Steuerung.Regelung_Modus.opti_Modus) THEN
	Zustand.Regelung_Modus := Steuerung.Regelung_Modus.opti;
ELSE
	Zustand.Regelung_Modus := Steuerung.Regelung_Modus.auto;
END_IF;
(* Priorisierung Regelung_Sollwert *)
IF(Steuerung.Regelung_Sollw.manu_Modus) THEN
	Zustand.Regelung_Sollw := Steuerung.Regelung_Sollw.manu;
ELSIF(Steuerung.Regelung_Sollw.opti_Modus) THEN
	Zustand.Regelung_Sollw := Steuerung.Regelung_Sollw.opti;
ELSE
	Zustand.Regelung_Sollw := Steuerung.Regelung_Sollw.auto;
END_IF;



IF (Zustand.Regelung_Modus_Anford )THEN
	Zustand.Regelung_Modus  :=E_Bel_Regelung_Modus_Lichtsensor ;
ELSE
	Zustand.Regelung_Modus := E_Bel_Regelung_Modus_P ;
END_IF

END_FUNCTION_BLOCK

// ---- POUs/Systeme/Sonstiges/Beleuchtung/FB_System_Bel_Zustandscheck.TcPOU
FUNCTION_BLOCK FB_System_Bel_Zustandscheck
VAR_IN_OUT
	Zustand					: ST_System_Bel_Zustand;
END_VAR
VAR_INPUT
	Steuerung				: ST_System_Bel_Steuerung;
	Parameter				: ST_System_Bel_Parameter;
END_VAR
VAR_OUTPUT
END_VAR
VAR
	Timer1: TON;
	Timer2: TON;
END_VAR

(*
	Stoerung_Code
		0:	*Allgemein Störung Beleuchtung (intern)
		1:	* Störung durch DALI-Lib
		2:	..
		3:
		4:
		5:
		6:
		7:

	Warnung_Code
		0:	*Allgemein Warnung Beleuchtung (intern)
		1:	keine Betriebsrückmeldung
		2:	keine Leistung
		3:	*Beleuchtung im Handbetrieb
		4:
		5:
		6:
		7:

	Freigabe_Code
		0:	*Freigabe durch Automatik entzogen
		1:	*Freigabe durch Manuell entzogen
		2:	*Freigabe durch Stoerung entzogen
		3: 	*Freigabe durch hohe Einschalthäufigkeiten entzogen
		4: 	*Freigabe durch zu hohe Rücklauf-Temperaturen entzogen
*)
Timer1(	IN := (Zustand.Betrieb_Anford <> Zustand.Betrieb),
		PT := T#1M,
		Q => Zustand.Warnung_Code.1
);

(* Warnung - keine Leistung im Betrieb nach 1 Minute *)
Timer2(	IN := Zustand.Leistung <= 0 AND Zustand.Betrieb_Anford = TRUE,
		PT := T#1M,
		Q => Zustand.Warnung_Code.2
);

END_FUNCTION_BLOCK
